PROGRAM MAIN
VAR
END_VAR

DistStationSensors();
DistStationControl();
TestStationSensors();
TestStationControl();
StationVisualProgram();

END_PROGRAM

(* stored: Version 1.1.0.1, ProductVersion 3.1.4018.5
   POU MAIN: Id {e73346dd-63f7-4b20-8cd4-ad522cfb0f53}, SpecialFunc None *)
